TYPE ST_GroupElement_HMI_Link EXTENDS ST_BaseGroupElement_HMI_Link :
STRUCT
	stGroupElement			: ST_GroupElement_HMI;

	stControlElement1		: ST_ControlElement_HMI_Link;
	stControlElement2		: ST_ControlElement_HMI_Link;
	stComponent1			: ST_Component_HMI_Link;
	stComponent2			: ST_Component_HMI_Link;
END_STRUCT
END_TYPE

(* stored: Version 1.1.0.1, ProductVersion 3.1.4024.15
   DUT ST_GroupElement_HMI_Link: Id {239f3496-eaed-4516-9961-8aaef0a09b2a} *)
